// TIA Portal V20 export
DATA_BLOCK "HmiInterface"   // DB19
// stored: Access Published, MemoryReserve 100, Namespace Unit1.Em2
   VAR
      em : "LAF_typeEmInterface";
      cm : "Unit1.Em2.typeCmHmiInterface";
      jrOutPnPLeft : "LER_typeSequenceInterface";
      jrOutPnPRight : "LER_typeSequenceInterface";
      emOverviewHomeCondition : "LER_typeEmOverviewHomeCondition";
      cmJROutPnPLeftSafetyPin : "LBC_typeDigitalSignalInterface";
      cmJROutPnPLeftJRDetect : "LBC_typeDigitalSignalInterface";
      cmJROutPnPRightSafetyPin : "LBC_typeDigitalSignalInterface";
      cmJROutPnPRightJRDetect : "LBC_typeDigitalSignalInterface";
      cmJROutPnPLeftAxisX : "LBC_typeAxis64PosInterface";
      cmJROutPnPLeftAxisZ : "LBC_typeAxis64PosInterface";
      cmJROutPnPRightAxisX : "LBC_typeAxis64PosInterface";
      cmJROutPnPRightAxisZ : "LBC_typeAxis64PosInterface";
      cmJROutPnPLeftClampOpenClose : "LBC_typeTwoWayActuatorInterface";
      cmJROutPnPRightClampOpenClose : "LBC_typeTwoWayActuatorInterface";
      intCondition : "Unit1.Em2.typeIntConditionHmiInterface";
   END_VAR
BEGIN
   cmJROutPnPLeftAxisX.configuration.setPositions[0]."name" := 'Wait';
   cmJROutPnPLeftAxisX.configuration.setPositions[1]."name" := 'Stack1 Load';
   cmJROutPnPLeftAxisX.configuration.setPositions[2]."name" := 'Stack2 Load';
   cmJROutPnPLeftAxisX.configuration.setPositions[3]."name" := 'Unload';
   cmJROutPnPLeftAxisX.configuration.setPositions[8]."name" := 'No Interference';
   cmJROutPnPLeftAxisX.configuration.setPositions[9]."name" := 'Stack1 Load Zone';
   cmJROutPnPLeftAxisX.configuration.setPositions[10]."name" := 'Stack2 Load Zone';
   cmJROutPnPLeftAxisX.configuration.setPositions[11]."name" := 'Unload Zone';
   cmJROutPnPLeftAxisZ.configuration.setPositions[0]."name" := 'Wait';
   cmJROutPnPLeftAxisZ.configuration.setPositions[1]."name" := 'Stack1 Load';
   cmJROutPnPLeftAxisZ.configuration.setPositions[2]."name" := 'Stack2 Load';
   cmJROutPnPLeftAxisZ.configuration.setPositions[3]."name" := 'Unload';
   cmJROutPnPLeftAxisZ.configuration.setPositions[8]."name" := 'No Interference Zone';
   cmJROutPnPRightAxisX.configuration.setPositions[0]."name" := 'Wait';
   cmJROutPnPRightAxisX.configuration.setPositions[1]."name" := 'Load';
   cmJROutPnPRightAxisX.configuration.setPositions[2]."name" := 'Unload';
   cmJROutPnPRightAxisX.configuration.setPositions[8]."name" := 'No Interference Zone';
   cmJROutPnPRightAxisX.configuration.setPositions[9]."name" := 'Load Zone';
   cmJROutPnPRightAxisX.configuration.setPositions[10]."name" := 'Unload Zone';
   cmJROutPnPRightAxisZ.configuration.setPositions[1]."name" := 'Load';
   cmJROutPnPRightAxisZ.configuration.setPositions[2]."name" := 'Unload';
   cmJROutPnPRightAxisZ.configuration.setPositions[8]."name" := 'No Interference Zone';
END_DATA_BLOCK
